FUNCTION_BLOCK AR2_R_TO_REAL (* Composite FB for convert AR2 to REAL *)
  (* Standard: 61499-2; Description: Copyright (c) 2024 HR Agrartechnik GmbH This program and the accompanying materials are made available under the terms of the Eclipse Public License 2.0 which is available at https://www.eclipse.org/legal/epl-2.0/ SPDX-License-Identifier: EPL-2.0 *)
  (* Version 1.0, 2024-04-24, Franz Höpfinger, HR Agrartechnik GmbH *)
  PACKAGE adapter::conversion::bidirectional;
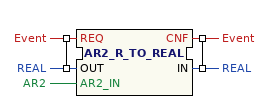
  EVENT_INPUT
    REQ WITH OUT; (* Request to Adapter *)
  END_EVENT
  EVENT_OUTPUT
    CNF WITH IN; (* Confirmation from Adapter *)
  END_EVENT
  VAR_INPUT
    OUT : REAL;
  END_VAR
  VAR_OUTPUT
    IN : REAL; (* Input data from Adapter *)
  END_VAR
  SOCKETS
    AR2_IN : adapter::types::bidirectional::AR2; (* Adapter Input *)
  END_SOCKETS
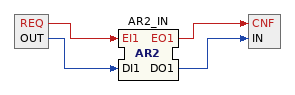
  EVENT_CONNECTIONS
    AR2_IN.EO1 TO CNF;
    REQ TO AR2_IN.EI1;
  END_CONNECTIONS
  DATA_CONNECTIONS
    AR2_IN.DO1 TO IN;
    OUT TO AR2_IN.DI1;
  END_CONNECTIONS
END_FUNCTION_BLOCK
